(*

short summary
=================
This interface provides assert statements for signed double integers (``DINT``)

.. <legal notes>

legal notes
=================
| SPDX-FileCopyrightText: © 2022 ekvip automation GmbH <info@ekvip.de>
| SPDX-License-Identifier: Apache-2.0
| For details check: Apache-2.0_

.. _Apache-2.0: https://www.apache.org/licenses/LICENSE-2.0

.. </legal notes>

methods
==================

*)

INTERFACE IDintAssertions EXTENDS __SYSTEM.IQueryInterface

(*

short summary
=================
This assertion method checks if the current value is equal to the expected value

.. <legal notes>

legal notes
=================
| SPDX-FileCopyrightText: © 2022 ekvip automation GmbH <info@ekvip.de>
| SPDX-License-Identifier: Apache-2.0
| For details check: Apache-2.0_

.. _Apache-2.0: https://www.apache.org/licenses/LICENSE-2.0

.. </legal notes>

parameters
=================

*)

METHOD valueIsEqualTo
VAR_INPUT
	(* current value to check *)
	currentValue	:DINT;
	(* expected value to compare *)
	expectedValue	:DINT;
	(* message if the assertion is false *)
	message			:AssertMessage;
END_VAR
END_METHOD

(*

short summary
=================
This assertion method checks if the current value is even

.. <legal notes>

legal notes
=================
| SPDX-FileCopyrightText: © 2022 ekvip automation GmbH <info@ekvip.de>
| SPDX-License-Identifier: Apache-2.0
| For details check: Apache-2.0_

.. _Apache-2.0: https://www.apache.org/licenses/LICENSE-2.0

.. </legal notes>

parameters
=================

*)

METHOD valueIsEven
VAR_INPUT
	(* current value to check *)
	currentValue	:DINT;
	(* message if the assertion is false *)
	message			:AssertMessage;
END_VAR
END_METHOD

(*

short summary
=================
This assertion method checks if the current value is greater than the less value

.. <legal notes>

legal notes
=================
| SPDX-FileCopyrightText: © 2022 ekvip automation GmbH <info@ekvip.de>
| SPDX-License-Identifier: Apache-2.0
| For details check: Apache-2.0_

.. _Apache-2.0: https://www.apache.org/licenses/LICENSE-2.0

.. </legal notes>

parameters
=================

*)

METHOD valueIsGreaterThan
VAR_INPUT
	(* current value to check *)
	currentValue	:DINT;
	(* less than lower limit *)
	lessValue		:DINT;
	(* message if the assertion is false *)
	message			:AssertMessage;
END_VAR
END_METHOD

(*

short summary
=================
This assertion method checks if the current value is inside a limit

.. attention:: 
	limits are included: ``valueIsInRangeOf(3, 3, 3)`` is a true assertion

.. <legal notes>

legal notes
=================
| SPDX-FileCopyrightText: © 2022 ekvip automation GmbH <info@ekvip.de>
| SPDX-License-Identifier: Apache-2.0
| For details check: Apache-2.0_

.. _Apache-2.0: https://www.apache.org/licenses/LICENSE-2.0

.. </legal notes>

parameters
=================

*)

METHOD valueIsInRangeOf
VAR_INPUT
	(* lower limit for the current value *)
	lowerLimit		:DINT;
	(* current value to check *)
	currentValue	:DINT;
	(* upper limit for the current value *)
	upperLimit		:DINT;
	(* message if the assertion is false *)
	message			:AssertMessage;
END_VAR
END_METHOD

(*

short summary
=================
This assertion method checks if the current value is less than the greater value

.. <legal notes>

legal notes
=================
| SPDX-FileCopyrightText: © 2022 ekvip automation GmbH <info@ekvip.de>
| SPDX-License-Identifier: Apache-2.0
| For details check: Apache-2.0_

.. _Apache-2.0: https://www.apache.org/licenses/LICENSE-2.0

.. </legal notes>

parameters
=================

*)

METHOD valueIsLessThan
VAR_INPUT
	(* current value to check *)
	currentValue	:DINT;
	(* greater than upper limit *)
	greaterValue	:DINT;
	(* message if the assertion is false *)
	message			:AssertMessage;
END_VAR
END_METHOD

(*

short summary
=================
This assertion method checks if the current value is less than or equal to the maximum value

.. <legal notes>

legal notes
=================
| SPDX-FileCopyrightText: © 2022 ekvip automation GmbH <info@ekvip.de>
| SPDX-License-Identifier: Apache-2.0
| For details check: Apache-2.0_

.. _Apache-2.0: https://www.apache.org/licenses/LICENSE-2.0

.. </legal notes>

parameters
=================

*)

METHOD valueIsMax
VAR_INPUT
	(* current value to check *)
	currentValue	:DINT;
	(* upper limit for the current value *)
	maximumValue	:DINT;
	(* message if the assertion is false *)
	message			:AssertMessage;
END_VAR
END_METHOD

(*

short summary
=================
This assertion method checks if the current value is greater than or equal to the minimum value

.. <legal notes>

legal notes
=================
| SPDX-FileCopyrightText: © 2022 ekvip automation GmbH <info@ekvip.de>
| SPDX-License-Identifier: Apache-2.0
| For details check: Apache-2.0_

.. _Apache-2.0: https://www.apache.org/licenses/LICENSE-2.0

.. </legal notes>

parameters
=================

*)

METHOD valueIsMin
VAR_INPUT
	(* current value to check *)
	currentValue	:DINT;
	(* lower limit for the current value *)
	minimumValue	:DINT;
	(* message if the assertion is false *)
	message			:AssertMessage;
END_VAR
END_METHOD

(*

short summary
=================
This assertion method checks if the current value is negative

.. <legal notes>

legal notes
=================
| SPDX-FileCopyrightText: © 2022 ekvip automation GmbH <info@ekvip.de>
| SPDX-License-Identifier: Apache-2.0
| For details check: Apache-2.0_

.. _Apache-2.0: https://www.apache.org/licenses/LICENSE-2.0

.. </legal notes>

parameters
=================

*)

METHOD valueIsNegative
VAR_INPUT
	(* current value to check *)
	currentValue	:DINT;
	(* message if the assertion is false *)
	message			:AssertMessage;
END_VAR
END_METHOD

(*

short summary
=================
This assertion method checks if the current value is not equal to the unexpected value

.. <legal notes>

legal notes
=================
| SPDX-FileCopyrightText: © 2022 ekvip automation GmbH <info@ekvip.de>
| SPDX-License-Identifier: Apache-2.0
| For details check: Apache-2.0_

.. _Apache-2.0: https://www.apache.org/licenses/LICENSE-2.0

.. </legal notes>

parameters
=================

*)

METHOD valueIsNotEqualTo
VAR_INPUT
	(* current value to check *)
	currentValue	:DINT;
	(* unexpected value to compare *)
	unexpectedValue	:DINT;
	(* message if the assertion is false *)
	message			:AssertMessage;
END_VAR
END_METHOD

(*

short summary
=================
This assertion method checks if the current value is odd

.. <legal notes>

legal notes
=================
| SPDX-FileCopyrightText: © 2022 ekvip automation GmbH <info@ekvip.de>
| SPDX-License-Identifier: Apache-2.0
| For details check: Apache-2.0_

.. _Apache-2.0: https://www.apache.org/licenses/LICENSE-2.0

.. </legal notes>

parameters
=================

*)

METHOD valueIsOdd
VAR_INPUT
	(* current value to check *)
	currentValue	:DINT;
	(* message if the assertion is false *)
	message			:AssertMessage;
END_VAR
END_METHOD

(*

short summary
=================
This assertion method checks if the current value is positve

.. <legal notes>

legal notes
=================
| SPDX-FileCopyrightText: © 2022 ekvip automation GmbH <info@ekvip.de>
| SPDX-License-Identifier: Apache-2.0
| For details check: Apache-2.0_

.. _Apache-2.0: https://www.apache.org/licenses/LICENSE-2.0

.. </legal notes>

parameters
=================

*)

METHOD valueIsPositive
VAR_INPUT
	(* current value to check *)
	currentValue	:DINT;
	(* message if the assertion is false *)
	message			:AssertMessage;
END_VAR
END_METHOD

END_INTERFACE

(* stored: Version 1.1.0.1, ProductVersion 3.1.4024.11
   Itf IDintAssertions: Id {eddb701f-08df-4387-967b-ff5fa864288f}
   Method valueIsEqualTo: Id {1cc31701-8bcf-47e2-9188-9a7bf5ecd72f}
   Method valueIsEven: Id {6937e816-b929-43d1-939b-c4cca93c6932}
   Method valueIsGreaterThan: Id {84179ab8-c65d-4397-8679-e6bd15e9a167}
   Method valueIsInRangeOf: Id {c7f89a88-d5cb-4a36-b810-7add7c8ba4fc}
   Method valueIsLessThan: Id {1a3e9da4-ec5a-456b-b3ab-e3b1f121407b}
   Method valueIsMax: Id {ec337916-ef8f-41af-a12d-19f0055e7ea5}
   Method valueIsMin: Id {61d6fad6-7729-4851-ae4c-9c62e4b3116f}
   Method valueIsNegative: Id {a5de6f61-bb99-42bb-84a6-6c832a28fa73}
   Method valueIsNotEqualTo: Id {ee021767-4f78-48e7-b8d0-aae624739861}
   Method valueIsOdd: Id {bb1bbc7b-ff22-42e5-a3de-edd1ba18ffe5}
   Method valueIsPositive: Id {13e96bb5-17f4-452f-9e89-b30f91d491d4} *)
